FUNCTION_BLOCK AxisMoveCommand IMPLEMENTS ITF_Command
VAR
	_reciever : ITF_Axis;
	_position : LREAL;
	_velocity : LREAL;
END_VAR

METHOD Execute : BOOL
IF _reciever <> 0 THEN
	_reciever.MoveToPosition(Position := _position, Velocity := _velocity);
END_IF
END_METHOD

PROPERTY MyAxis : ITF_Axis
GET
MyAxis := _reciever;
END_GET
SET
_reciever := MyAxis;
END_SET
END_PROPERTY

PROPERTY Position : LREAL
GET
Position := _position;
END_GET
SET
_position := Position;
END_SET
END_PROPERTY

PROPERTY Velocity : LREAL
GET
Velocity := _velocity;
END_GET
SET
_velocity := Velocity;
END_SET
END_PROPERTY

END_FUNCTION_BLOCK

(* stored: Version 1.1.0.1, ProductVersion 3.1.4024.12
   POU AxisMoveCommand: Id {94afdd16-a13b-48ee-b5b1-240dd1446e8d}, SpecialFunc None
   Method Execute: Id {b614749c-f6db-4941-9b5d-24cd04244641}
   Property MyAxis: Id {31f54a33-00ef-4d7a-9c89-4638d26d502b}
   Get Get: Id {8103b9f1-c5e1-4b51-b8a6-f9d492a3c245}
   Set Set: Id {7814ae0c-452a-478a-9b94-271637a1eda2}
   Property Position: Id {26356e8c-188d-4c0c-82e1-df3d8758c5b8}
   Get Get: Id {337f572a-26c6-4235-b2e2-119458aa2251}
   Set Set: Id {2ae4f3ac-6be1-4de8-9557-eb9422c565d6}
   Property Velocity: Id {4ccb7d0b-ce3a-4da2-ab60-337ede9c4be1}
   Get Get: Id {efa7ef84-5a5d-48ee-8fee-4796a5f85932}
   Set Set: Id {2f85ea6b-0c0c-4bfc-a401-744e27d8cb46} *)
